(* IEC 61131-3 sources: RL_MAR/experiments/results/ablation/RL_MAR_DeepSeek-V3.2_full (part 2) *)

(* ---- med_62.st ---- *)
FUNCTION_BLOCK FB_PedestrianTrafficLight
VAR_INPUT
    pedBtnPress : BOOL;
END_VAR

VAR_OUTPUT
    carLightIsGreen : BOOL;
    pedLightIsGreen : BOOL;
    TimeCounter : INT;
END_VAR

VAR
    buttonPressedBefore : BOOL := FALSE;
    currentState : INT := 0;
    nextState : INT := 0;
END_VAR

CASE currentState OF
    0:
        carLightIsGreen := TRUE;
        pedLightIsGreen := FALSE;
        TimeCounter := 0;

        IF pedBtnPress AND NOT buttonPressedBefore THEN
            buttonPressedBefore := TRUE;
            nextState := 1;
        ELSE
            nextState := 0;
        END_IF;

    1:
        carLightIsGreen := FALSE;
        pedLightIsGreen := FALSE;
        TimeCounter := TimeCounter + 1;

        IF TimeCounter >= 10 THEN
            nextState := 2;
        ELSE
            nextState := 1;
        END_IF;

    2:
        carLightIsGreen := FALSE;
        pedLightIsGreen := TRUE;
        TimeCounter := TimeCounter + 1;

        IF TimeCounter >= 40 THEN
            nextState := 3;
        ELSE
            nextState := 2;
        END_IF;

    3:
        carLightIsGreen := FALSE;
        pedLightIsGreen := FALSE;
        TimeCounter := TimeCounter + 1;

        IF TimeCounter >= 50 THEN
            buttonPressedBefore := FALSE;
            nextState := 0;
        ELSE
            nextState := 3;
        END_IF;

    ELSE
        nextState := 0;
END_CASE;

currentState := nextState;

END_FUNCTION_BLOCK;

(* ---- med_63.st ---- *)
FUNCTION_BLOCK Automated_Parking_Controller
VAR_INPUT
    EntryGateSensor : BOOL; (* Sensor input for entry gate *)
    ExitGateSensor : BOOL; (* Sensor input for exit gate *)
    CarDetected : BOOL; (* Sensor input for car detection *)
END_VAR

VAR_OUTPUT
    ParkingSpaceNumber : INT := 0; (* Allocated parking space number *)
    RetrievalInProgress : BOOL := FALSE; (* Flag for car retrieval in progress *)
END_VAR

VAR
    ParkingSpaces : ARRAY[1..100] OF BOOL; (* Parking space status: TRUE=Occupied, FALSE=Available *)
    i : INT; (* Loop counter *)
    SpaceToRetrieve : INT := 0; (* Parking space number to retrieve *)
    RetrievalComplete : BOOL := FALSE; (* Internal flag for retrieval completion *)
END_VAR

METHOD MoveCarToExitGate : BOOL
VAR_INPUT
    SpaceNumber : INT;
END_VAR
BEGIN
    // Simulate car movement to exit gate
    // In a real system, this would control actuators, motors, etc.
    // For now, return TRUE to indicate successful movement
    MoveCarToExitGate := TRUE;
END_METHOD

// Main logic
IF NOT RetrievalInProgress THEN
    // Entry gate management
    IF EntryGateSensor THEN
        // Find first available parking space
        ParkingSpaceNumber := 0;
        FOR i := 1 TO 100 DO
            IF NOT ParkingSpaces[i] THEN
                ParkingSpaceNumber := i;
                ParkingSpaces[i] := TRUE;
                EXIT;
            END_IF;
        END_FOR;
    END_IF;
END_IF;

// Car retrieval management
IF CarDetected AND NOT RetrievalInProgress THEN
    RetrievalInProgress := TRUE;
    SpaceToRetrieve := ParkingSpaceNumber;
    RetrievalComplete := FALSE;
END_IF;

IF RetrievalInProgress THEN
    IF NOT RetrievalComplete THEN
        // Execute car movement to exit gate
        RetrievalComplete := MoveCarToExitGate(SpaceToRetrieve);
    ELSE
        // Wait for exit gate sensor to confirm car has left
        IF ExitGateSensor THEN
            // Mark parking space as available
            IF SpaceToRetrieve >= 1 AND SpaceToRetrieve <= 100 THEN
                ParkingSpaces[SpaceToRetrieve] := FALSE;
            END_IF;

            // Reset outputs
            ParkingSpaceNumber := 0;
            RetrievalInProgress := FALSE;
            SpaceToRetrieve := 0;
            RetrievalComplete := FALSE;
        END_IF;
    END_IF;
END_IF;

// Exit gate management (for normal exits without retrieval request)
IF ExitGateSensor AND NOT RetrievalInProgress AND ParkingSpaceNumber > 0 THEN
    // Mark current parking space as available
    IF ParkingSpaceNumber >= 1 AND ParkingSpaceNumber <= 100 THEN
        ParkingSpaces[ParkingSpaceNumber] := FALSE;
    END_IF;
    ParkingSpaceNumber := 0;
END_IF;

END_FUNCTION_BLOCK

(* ---- med_64.st ---- *)
FUNCTION_BLOCK BakeryOvenControl
VAR_INPUT
    TemperatureSensor : REAL; (* Sensor input for oven temperature *)
    HumiditySensor : REAL; (* Sensor input for oven humidity *)
END_VAR

VAR_OUTPUT
    HeatingElement : BOOL; (* Control signal for heating element *)
    CoolingElement : BOOL; (* Control signal for cooling element *)
    HumidityControl : BOOL; (* Control signal for humidity system *)
    DehumidityControl : BOOL; (* Control signal for dehumidification *)
END_VAR

VAR
    OvenTemperature : REAL := 180.0; (* Current oven temperature setpoint *)
    OvenHumidity : REAL := 60.0; (* Current oven humidity setpoint *)
    BakingTime : TIME := T#30M0S; (* Baking time setpoint *)
    OvenStatus : BOOL := FALSE; (* Oven status: TRUE=On, FALSE=Off *)
    HeatingThreshold : REAL := 2.0; (* Temperature control threshold *)
    HumidityThreshold : REAL := 5.0; (* Humidity control threshold *)
    TimerInstance : TON; (* Timer instance for 1-second decrement *)
    TimerPulse : BOOL := FALSE; (* Pulse for timer decrement *)
    InternalBakingTime : TIME := T#0S; (* Internal copy of baking time *)
END_VAR

(* Main logic body begins here *)

(* Timer for 1-second pulse generation *)
TimerInstance(IN := OvenStatus AND (InternalBakingTime > T#0S), PT := T#1S);
TimerPulse := TimerInstance.Q;

(* Decrement baking timer when oven is on and timer pulse is active *)
IF OvenStatus AND TimerPulse THEN
    IF InternalBakingTime > T#0S THEN
        InternalBakingTime := InternalBakingTime - T#1S;
    END_IF;
END_IF;

(* Reset internal timer when oven turns off *)
IF NOT OvenStatus THEN
    InternalBakingTime := BakingTime;
END_IF;

(* Main control logic - only active when oven is on and timer not expired *)
IF OvenStatus AND (InternalBakingTime > T#0S) THEN
    (* Temperature control logic *)
    IF TemperatureSensor < (OvenTemperature - HeatingThreshold) THEN
        HeatingElement := TRUE;
        CoolingElement := FALSE;
    ELSIF TemperatureSensor > (OvenTemperature + HeatingThreshold) THEN
        HeatingElement := FALSE;
        CoolingElement := TRUE;
    ELSE
        HeatingElement := FALSE;
        CoolingElement := FALSE;
    END_IF;

    (* Humidity control logic *)
    IF HumiditySensor < (OvenHumidity - HumidityThreshold) THEN
        HumidityControl := TRUE;
        DehumidityControl := FALSE;
    ELSIF HumiditySensor > (OvenHumidity + HumidityThreshold) THEN
        HumidityControl := FALSE;
        DehumidityControl := TRUE;
    ELSE
        HumidityControl := FALSE;
        DehumidityControl := FALSE;
    END_IF;

(* Oven off or timer expired - turn off all outputs *)
ELSE
    HeatingElement := FALSE;
    CoolingElement := FALSE;
    HumidityControl := FALSE;
    DehumidityControl := FALSE;

    (* Auto-shutdown when timer expires *)
    IF (InternalBakingTime <= T#0S) AND OvenStatus THEN
        OvenStatus := FALSE;
    END_IF;
END_IF;

END_FUNCTION_BLOCK;

(* ---- med_65.st ---- *)
FUNCTION_BLOCK TheaterControl
VAR_INPUT
    StartButton : BOOL; (* Input for starting a performance *)
    StopButton : BOOL; (* Input for stopping a performance *)
    SceneNumber : INT; (* Input for selecting the scene or act *)
END_VAR

VAR_OUTPUT
    LightingControl : BOOL; (* Output for controlling lighting *)
    SoundControl : BOOL; (* Output for controlling sound *)
    PerformanceInProgress : BOOL; (* Indicator for an ongoing performance *)
END_VAR

VAR
    CurrentState : INT := 1; (* 1=IDLE, 2=ACTIVE, 3=STOP *)
    NextState : INT;
END_VAR

(* State Machine Logic *)
CASE CurrentState OF
    1: (* IDLE State *)
        LightingControl := FALSE;
        SoundControl := FALSE;
        PerformanceInProgress := FALSE;

        IF StopButton THEN
            NextState := 3;
        ELSIF StartButton AND NOT PerformanceInProgress THEN
            IF (SceneNumber >= 1) AND (SceneNumber <= 3) THEN
                NextState := 2;
            ELSE
                NextState := 3;
            END_IF;
        ELSE
            NextState := 1;
        END_IF;

    2: (* ACTIVE State *)
        LightingControl := TRUE;
        SoundControl := TRUE;
        PerformanceInProgress := TRUE;

        IF StopButton THEN
            NextState := 3;
        ELSE
            NextState := 2;
        END_IF;

    3: (* STOP State *)
        LightingControl := FALSE;
        SoundControl := FALSE;
        PerformanceInProgress := FALSE;
        NextState := 1;

END_CASE;

(* State Transition *)
CurrentState := NextState;

END_FUNCTION_BLOCK;

(* ---- med_66.st ---- *)
FUNCTION_BLOCK ElevatorControl
VAR_INPUT
    CurrentPos : INT;
    RequestedPos : INT;
    ButtonPressed : BOOL;
END_VAR

VAR_OUTPUT
    MotorMovingUp : BOOL;
    MotorMovingDown : BOOL;
    DoorIsOpen : BOOL;
END_VAR

VAR
    bMovementInitiated : BOOL := FALSE;
END_VAR

(* Main logic body begins here *)

(* Reset outputs on each cycle *)
MotorMovingUp := FALSE;
MotorMovingDown := FALSE;
DoorIsOpen := FALSE;

(* Handle button press to initiate movement *)
IF ButtonPressed THEN
    bMovementInitiated := TRUE;
    DoorIsOpen := FALSE;
END_IF;

(* Determine movement direction and handle state transitions *)
IF bMovementInitiated THEN
    IF CurrentPos < RequestedPos THEN
        (* Move up *)
        MotorMovingUp := TRUE;
        MotorMovingDown := FALSE;
        DoorIsOpen := FALSE;
    ELSIF CurrentPos > RequestedPos THEN
        (* Move down *)
        MotorMovingUp := FALSE;
        MotorMovingDown := TRUE;
        DoorIsOpen := FALSE;
    ELSE
        (* Reached destination *)
        MotorMovingUp := FALSE;
        MotorMovingDown := FALSE;
        DoorIsOpen := TRUE;
        bMovementInitiated := FALSE;
    END_IF;
ELSE
    (* Stationary at requested floor *)
    IF CurrentPos = RequestedPos THEN
        DoorIsOpen := TRUE;
    END_IF;
END_IF;

END_FUNCTION_BLOCK;

(* ---- med_67.st ---- *)
FUNCTION_BLOCK FB_FactorialCalculator
VAR_INPUT
    X : INT;
END_VAR

VAR_OUTPUT
    FactorialResult : INT;
    FactorialGoodResult : INT;
END_VAR

VAR
    tempGoodResult : INT;
    tempResult : INT;
END_VAR

// Main logic
IF (X >= -3) AND (X <= 3) THEN
    // Calculate FactorialGoodResult = X * X * X * X
    tempGoodResult := X * X;
    tempGoodResult := tempGoodResult * X;
    tempGoodResult := tempGoodResult * X;
    FactorialGoodResult := tempGoodResult;

    // Calculate FactorialResult
    IF FactorialGoodResult > 1 THEN
        tempResult := FactorialGoodResult - 1;
        FactorialResult := FactorialGoodResult * tempResult;
    ELSE
        FactorialResult := FactorialGoodResult;
    END_IF;
ELSE
    // X is outside range [-3, 3]
    FactorialGoodResult := 0;
    FactorialResult := 1;
END_IF;
END_FUNCTION_BLOCK

(* ---- med_68.st ---- *)
FUNCTION_BLOCK SignalControl
VAR_INPUT
    Int1 : BOOL;
    Int2 : BOOL;
    Int3 : BOOL;
    Int4 : BOOL;
    Int5 : BOOL;
    Int6 : BOOL;
    Int7 : BOOL;
    Int8 : BOOL;
    IntAn1 : UINT;
    IntAn2 : UINT;
    IntAn3 : UINT;
    IntAn4 : UINT;
    IntAn5 : UINT;
    IntAn6 : UINT;
    IntAn7 : UINT;
    IntAn8 : UINT;
    Marca2 : BOOL;
END_VAR

VAR_OUTPUT
    Out1 : BOOL;
    Out2 : BOOL;
    Out3 : BOOL;
    Out4 : BOOL;
    Out5 : BOOL;
    Out6 : BOOL;
    Out7 : BOOL;
    Out8 : BOOL;
    OutAn1 : UINT;
    OutAn2 : UINT;
    OutAn3 : UINT;
    OutAn4 : UINT;
    OutAn5 : UINT;
    OutAn6 : UINT;
    OutAn7 : UINT;
    OutAn8 : UINT;
END_VAR

VAR
    Marca1 : BOOL;
    GT51_OUT : BOOL;
    GT56_OUT : BOOL;
    GT57_OUT : BOOL;
    GT62_OUT : BOOL;
END_VAR

    (* Logic for Marca1 flag *)
    IF NOT Marca2 AND ((Marca1 OR NOT Out1) AND Int1) THEN
        Marca1 := TRUE;
    ELSE
        Marca1 := FALSE;
    END_IF;

    (* Latch behavior for Out1 *)
    IF NOT Marca2 AND (Marca1 OR Out1) THEN
        Out1 := TRUE;
    ELSE
        Out1 := FALSE;
    END_IF;

    (* Direct Boolean pass-through *)
    Out2 := Int2;
    Out3 := Int3;
    Out4 := Int4;

    (* Direct unsigned integer pass-through *)
    OutAn1 := IntAn1;
    OutAn2 := IntAn2;
    OutAn3 := IntAn3;
    OutAn4 := IntAn4;

    (* Conditional outputs with comparison results *)
    GT51_OUT := (IntAn5 > 1000);
    GT56_OUT := (IntAn6 > 1000);
    GT57_OUT := (IntAn7 > 1000);
    GT62_OUT := (IntAn8 > 1000);

    (* Conditional output logic for Out5 *)
    IF GT51_OUT AND NOT Int5 THEN
        Out5 := TRUE;
    ELSE
        Out5 := FALSE;
    END_IF;

    (* Conditional output logic for Out6 *)
    IF GT56_OUT AND NOT Int6 THEN
        Out6 := TRUE;
    ELSE
        Out6 := FALSE;
    END_IF;

    (* Conditional output logic for Out7 *)
    IF GT57_OUT AND NOT Int7 THEN
        Out7 := TRUE;
    ELSE
        Out7 := FALSE;
    END_IF;

    (* Conditional output logic for Out8 *)
    IF GT62_OUT AND NOT Int8 THEN
        Out8 := TRUE;
    ELSE
        Out8 := FALSE;
    END_IF;

    (* Pass through remaining analog values *)
    OutAn5 := IntAn5;
    OutAn6 := IntAn6;
    OutAn7 := IntAn7;
    OutAn8 := IntAn8;

END_FUNCTION_BLOCK;

(* ---- med_69.st ---- *)
FUNCTION_BLOCK FB_ValueOut
VAR_INPUT
    valueIn : INT;
    conf : UINT;
END_VAR

VAR_OUTPUT
    ValueOut : INT;
END_VAR

VAR
    tempResult : INT;
END_VAR

(* Main logic body *)
CASE conf OF
    1, 2:
        tempResult := valueIn / 10;
        IF tempResult < 0 THEN
            ValueOut := 0;
        ELSE
            ValueOut := tempResult;
        END_IF;

    3:
        IF valueIn = 0 THEN
            ValueOut := 0;
        ELSIF valueIn = 300 THEN
            ValueOut := 163;
        ELSIF valueIn = 600 THEN
            ValueOut := 331;
        ELSE
            ValueOut := 0;
        END_IF;

    6, 7:
        IF valueIn = 100 THEN
            ValueOut := 319;
        ELSE
            ValueOut := 0;
        END_IF;

    ELSE
        ValueOut := 0;
END_CASE;

END_FUNCTION_BLOCK;

(* ---- med_70.st ---- *)
FUNCTION_BLOCK EggIncubatorControl
VAR_INPUT
    StartButton : BOOL; (* Input for starting the incubation process *)
    StopButton : BOOL; (* Input for stopping the incubation process *)
    TemperatureSensor : REAL; (* Input for temperature reading in °C *)
    HumiditySensor : REAL; (* Input for humidity reading in % *)
END_VAR

VAR_OUTPUT
    HeatingElement : BOOL; (* Output for controlling the heating element *)
    Humidifier : BOOL; (* Output for controlling the humidifier *)
    EggTurningMotor : BOOL; (* Output for controlling the egg turning motor *)
    IncubationInProgress : BOOL; (* Indicator for an ongoing incubation process *)
END_VAR

VAR
    TargetTemperature : REAL; (* Target temperature in °C *)
    TargetHumidity : REAL; (* Target humidity in % *)
    TurnIntervalSeconds : INT; (* Interval for turning eggs (1 hour in seconds) *)
    TurnTimerSeconds : INT; (* Timer for egg turning cycle in seconds *)
END_VAR

(* Initialize control parameters *)
TargetTemperature := 37.5;
TargetHumidity := 50.0;
TurnIntervalSeconds := 3600;

(* Start/Stop Control *)
IF StartButton AND NOT IncubationInProgress THEN
    IncubationInProgress := TRUE;
END_IF;

IF StopButton THEN
    IncubationInProgress := FALSE;
    HeatingElement := FALSE;
    Humidifier := FALSE;
    EggTurningMotor := FALSE;
    TurnTimerSeconds := 0;
END_IF;

(* Temperature Control *)
IF TemperatureSensor < TargetTemperature THEN
    HeatingElement := TRUE;
ELSE
    HeatingElement := FALSE;
END_IF;

(* Humidity Control *)
IF HumiditySensor < TargetHumidity THEN
    Humidifier := TRUE;
ELSE
    Humidifier := FALSE;
END_IF;

(* Egg Turning Cycle *)
IF IncubationInProgress THEN
    TurnTimerSeconds := TurnTimerSeconds + 1;
    IF TurnTimerSeconds >= TurnIntervalSeconds THEN
        EggTurningMotor := NOT EggTurningMotor;
        TurnTimerSeconds := 0;
    END_IF;
END_IF;

END_FUNCTION_BLOCK;

(* ---- med_71.st ---- *)
FUNCTION_BLOCK FB_Fibonacci_Calculator
VAR_INPUT
    N : DINT := 5;
END_VAR
VAR_OUTPUT
    O : DINT := 1;
END_VAR
VAR
    F1 : DINT := 1;
    F2 : DINT := 1;
    CNT : DINT := 2;
    Temp : DINT;
END_VAR

// Handle edge cases: N <= 2 returns 1
IF N <= 2 THEN
    O := 1;
    RETURN;
END_IF;

// Initialize for calculation
F1 := 1;
F2 := 1;
CNT := 2;

// Calculate Fibonacci sequence up to N-th term
WHILE CNT < N DO
    // Check for potential overflow before calculation
    IF (F1 > 32767 - F2) THEN
        // Saturation: if sum would exceed 32767, saturate to 32767
        O := 32767;
        RETURN;
    END_IF;

    // Calculate next Fibonacci number
    Temp := F1 + F2;
    F1 := F2;
    F2 := Temp;
    CNT := CNT + 1;
END_WHILE;

// Set output to the N-th Fibonacci number
O := F2;

// Final saturation check (in case F2 already exceeded 32767)
IF O > 32767 THEN
    O := 32767;
END_IF;

END_FUNCTION_BLOCK

(* ---- med_72.st ---- *)
FUNCTION_BLOCK DigitalSignageManagement
VAR_INPUT
    DisplayLocations : ARRAY[1..10] OF BOOL;
    ContentSource : ARRAY[1..10] OF INT;
END_VAR

VAR_OUTPUT
    CurrentContent : ARRAY[1..10] OF INT;
END_VAR

VAR
    i : INT;
END_VAR

FOR i := 1 TO 10 DO
    IF DisplayLocations[i] THEN
        CASE ContentSource[i] OF
            1:
                CurrentContent[i] := 1;
            2:
                CurrentContent[i] := 2;
            3:
                CurrentContent[i] := 3;
            ELSE
                CurrentContent[i] := 0;
        END_CASE;
    ELSE
        CurrentContent[i] := 0;
    END_IF;
END_FOR;

END_FUNCTION_BLOCK;

(* ---- med_73.st ---- *)
FUNCTION_BLOCK RoboticWeldingSystem
    VAR_INPUT
        RobotArm1Ready : BOOL; (* Input for robot arm 1 ready status *)
        RobotArm2Ready : BOOL; (* Input for robot arm 2 ready status *)
        WeldingGunReady : BOOL; (* Input for welding gun ready status *)
        StartButton : BOOL; (* Input for start button press *)
        StopButton : BOOL; (* Input for stop button press *)
    END_VAR

    VAR_OUTPUT
        WeldingTrigger : BOOL; (* Output to trigger welding *)
        WeldingComplete : BOOL; (* Output indicating welding completion *)
    END_VAR

    VAR
        weldingActive : BOOL;
    END_VAR

    IF StopButton THEN
        weldingActive := FALSE;
        WeldingTrigger := FALSE;
        WeldingComplete := TRUE;
    ELSE
        IF NOT weldingActive AND RobotArm1Ready AND RobotArm2Ready AND WeldingGunReady AND StartButton THEN
            weldingActive := TRUE;
            WeldingTrigger := TRUE;
            WeldingComplete := FALSE;
        ELSIF weldingActive THEN
            WeldingTrigger := TRUE;
            WeldingComplete := FALSE;
        ELSE
            WeldingTrigger := FALSE;
            WeldingComplete := TRUE;
        END_IF;
    END_IF;
END_FUNCTION_BLOCK

(* ---- med_74.st ---- *)
FUNCTION_BLOCK TrafficManagementSystem
VAR_INPUT
    VehicleCount1 : INT; (* Input for vehicle count at intersection 1 *)
    VehicleCount2 : INT; (* Input for vehicle count at intersection 2 *)
    VehicleCount3 : INT; (* Input for vehicle count at intersection 3 *)
    VehicleCount4 : INT; (* Input for vehicle count at intersection 4 *)
END_VAR

VAR_OUTPUT
    TrafficLight1 : BOOL; (* Output for traffic light at intersection 1 *)
    TrafficLight2 : BOOL; (* Output for traffic light at intersection 2 *)
    TrafficLight3 : BOOL; (* Output for traffic light at intersection 3 *)
    TrafficLight4 : BOOL; (* Output for traffic light at intersection 4 *)
END_VAR

VAR
    (* No internal variables needed for this simplified implementation *)
END_VAR

(* Main logic for intersection pair 1 (Intersections 1 and 2) *)
IF VehicleCount1 > VehicleCount2 THEN
    TrafficLight1 := TRUE;
    TrafficLight2 := FALSE;
ELSIF VehicleCount1 < VehicleCount2 THEN
    TrafficLight1 := FALSE;
    TrafficLight2 := TRUE;
ELSE
    TrafficLight1 := FALSE;
    TrafficLight2 := FALSE;
END_IF;

(* Main logic for intersection pair 2 (Intersections 3 and 4) *)
IF VehicleCount3 > VehicleCount4 THEN
    TrafficLight3 := TRUE;
    TrafficLight4 := FALSE;
ELSIF VehicleCount3 < VehicleCount4 THEN
    TrafficLight3 := FALSE;
    TrafficLight4 := TRUE;
ELSE
    TrafficLight3 := FALSE;
    TrafficLight4 := FALSE;
END_IF;

END_FUNCTION_BLOCK;

(* ---- med_75.st ---- *)
FUNCTION_BLOCK HomeBrewingSystem
VAR_INPUT
    TemperatureSensor : REAL; (* Input for temperature measurement (°C) *)
    WaterFlowSensor : REAL; (* Input for water flow measurement (L/min) *)
    BrewingStartTime : TIME; (* Input for brewing process start time *)
    BrewingDuration : TIME; (* Input for total brewing duration *)
END_VAR

VAR_OUTPUT
    HeatingElement : BOOL; (* Output to control heating element *)
    AgitationMotor : BOOL; (* Output to control agitation motor *)
    HopsDispenser : BOOL; (* Output to control hops dispenser *)
    FermentationTank : BOOL; (* Output to control fermentation tank *)
END_VAR

VAR
    ElapsedTime : TIME;
    HopsTriggerTime : TIME := T#5h;
    FermentationTriggerTime : TIME := T#48h;
END_VAR

(* Main logic body *)
ElapsedTime := BrewingDuration;

(* Temperature control: heating element ON when temperature is below 65°C *)
HeatingElement := TemperatureSensor < 65.0;

(* Agitation motor control: motor ON when water flow exceeds 0.5 L/min *)
AgitationMotor := WaterFlowSensor > 0.5;

(* Hops dispenser: activate after 5 hours of brewing *)
HopsDispenser := ElapsedTime >= HopsTriggerTime;

(* Fermentation tank transfer: activate after 48 hours of brewing *)
FermentationTank := ElapsedTime >= FermentationTriggerTime;

END_FUNCTION_BLOCK;

(* ---- med_76.st ---- *)
FUNCTION_BLOCK MultimediaArtInstallationControl
VAR_INPUT
    MotionSensor : BOOL; (* Motion detection input *)
    AudioTrack : BOOL; (* Selected audio track *)
    VisualContent : BOOL; (* Selected visual content *)
END_VAR

VAR_OUTPUT
    LightingControl : BOOL; (* Lighting control output *)
    AudioControl : BOOL; (* Audio playback control *)
    VisualControl : BOOL; (* Visual display control *)
    ActivationTimer : INT; (* Timer for activation duration *)
END_VAR

VAR
    bMotionDetectedPrev : BOOL; (* Previous state of motion sensor *)
    bElementsActive : BOOL; (* State of all multimedia elements *)
END_VAR

(* Main logic *)
IF MotionSensor THEN
    (* Motion detected: activate all elements *)
    LightingControl := TRUE;
    AudioControl := AudioTrack; (* Only activate if audio track is selected *)
    VisualControl := VisualContent; (* Only activate if visual content is selected *)
    bElementsActive := TRUE;

    (* Increment activation timer up to 300 seconds *)
    IF ActivationTimer < 300 THEN
        ActivationTimer := ActivationTimer + 1;
    END_IF;

    (* Store current motion state for edge detection *)
    bMotionDetectedPrev := TRUE;

ELSE
    (* No motion detected: deactivate all elements *)
    LightingControl := FALSE;
    AudioControl := FALSE;
    VisualControl := FALSE;
    bElementsActive := FALSE;

    (* Reset timer when no motion is detected *)
    ActivationTimer := 0;

    (* Store current motion state for edge detection *)
    bMotionDetectedPrev := FALSE;
END_IF;

(* Safety protocol: Ensure elements are only active when motion is detected *)
IF NOT MotionSensor AND bElementsActive THEN
    LightingControl := FALSE;
    AudioControl := FALSE;
    VisualControl := FALSE;
    bElementsActive := FALSE;
    ActivationTimer := 0;
END_IF;

END_FUNCTION_BLOCK

(* ---- med_77.st ---- *)
FUNCTION_BLOCK OutdoorLEDLightingControl
VAR_INPUT
    AmbientLight : REAL; (* 环境光传感器输入 *)
    MotionSensor : BOOL; (* 运动传感器输入 *)
    EnergySaving : BOOL; (* 节能模式开关 *)
END_VAR

VAR_OUTPUT
    Light : BOOL; (* LED照明控制输出 *)
    EnergyMode : BOOL; (* 节能模式状态输出 *)
END_VAR

VAR
    (* No internal variables needed for this simple logic *)
END_VAR

(* Main logic body *)
IF MotionSensor THEN
    (* Motion Detection Override: Highest priority *)
    Light := TRUE;
    EnergyMode := FALSE; (* Override: deactivate energy-saving mode *)
ELSE
    (* No motion detected: evaluate ambient light and energy-saving mode *)
    IF (AmbientLight < 50.0) AND (NOT EnergySaving) THEN
        Light := TRUE;
    ELSE
        Light := FALSE;
    END_IF;

    (* Energy mode status reflects the input *)
    EnergyMode := EnergySaving;
END_IF;

END_FUNCTION_BLOCK;

(* ---- med_78.st ---- *)
FUNCTION_BLOCK RetractableRoofControl
    VAR_INPUT
        RainSensor : BOOL; (* Rain detection *)
        WindSensor : BOOL; (* Wind detection *)
        TemperatureSensor : REAL; (* Temperature input *)
    END_VAR

    VAR_OUTPUT
        RoofMotor : BOOL; (* Motor control *)
    END_VAR

    VAR
        TemperatureThreshold : REAL := 20.0;
    END_VAR

    (* Main logic body begins here *)
    IF RainSensor AND WindSensor THEN
        RoofMotor := TRUE;
    ELSIF RainSensor THEN
        RoofMotor := TRUE;
    ELSIF TemperatureSensor < TemperatureThreshold THEN
        RoofMotor := TRUE;
    ELSE
        RoofMotor := FALSE;
    END_IF;

END_FUNCTION_BLOCK;

(* ---- med_79.st ---- *)
FUNCTION_BLOCK CapsuleFillingMachineControl
VAR_INPUT
    CapsuleWeight : REAL;        (* Current capsule weight *)
    TargetWeight : REAL;         (* Target weight to achieve *)
    CapsuleInPosition : BOOL;    (* Capsule position sensor *)
    HopperEmpty : BOOL;          (* Hopper empty sensor *)
END_VAR
VAR_OUTPUT
    FeederMotor : BOOL;          (* Feeder motor control *)
    FillingMotor : BOOL;         (* Filling motor control *)
    ConveyorMotor : BOOL;        (* Conveyor motor control *)
    FillingInProgress : BOOL;    (* Filling status *)
    ErrorCode : INT;             (* Error indication: 0=OK, 1=CapsuleNotDetected, 2=FillingTimeout *)
END_VAR
VAR
    (* State machine *)
    CurrentState : INT := 0;     (* 0=IDLE, 1=CONVEYING, 2=FILLING, 3=CONVEYING_OUT *)

    (* Timers *)
    ConveyorTimer : TON;
    FillingTimer : TON;
    ConveyOutTimer : TON;

    (* Timing parameters *)
    ConveyorTime : TIME := T#2S;
    MaxFillingTime : TIME := T#10S;
    ConveyOutTime : TIME := T#1S;

    (* Error detection *)
    CapsuleDetectTimeout : TON;
    CapsuleDetectTime : TIME := T#5S;

    (* Filling control *)
    WeightTolerance : REAL := 0.1;
    FillingSpeed : REAL := 0.0;
    LastCapsuleWeight : REAL := 0.0;

    (* Internal flags *)
    CapsuleDetected : BOOL := FALSE;
    FillingComplete : BOOL := FALSE;
    ErrorFlag : BOOL := FALSE;
END_VAR

(* Safety Check: Hopper Empty *)
IF HopperEmpty THEN
    FeederMotor := FALSE;
    FillingMotor := FALSE;
    ConveyorMotor := FALSE;
    FillingInProgress := FALSE;
    ErrorCode := 0;
    CurrentState := 0;
    RETURN;
END_IF;

(* Weight Validation: Initial Check *)
IF CapsuleWeight >= TargetWeight AND NOT FillingInProgress THEN
    FeederMotor := FALSE;
    FillingMotor := FALSE;
    ConveyorMotor := FALSE;
    FillingInProgress := FALSE;
    ErrorCode := 0;
    CurrentState := 0;
    RETURN;
END_IF;

(* State Machine Execution *)
CASE CurrentState OF
    0: (* IDLE *)
        FeederMotor := TRUE;
        FillingMotor := FALSE;
        ConveyorMotor := FALSE;
        FillingInProgress := FALSE;
        FillingComplete := FALSE;
        ErrorFlag := FALSE;
        ErrorCode := 0;

        (* Reset timers *)
        ConveyorTimer(IN:=FALSE, PT:=ConveyorTime);
        FillingTimer(IN:=FALSE, PT:=MaxFillingTime);
        ConveyOutTimer(IN:=FALSE, PT:=ConveyOutTime);
        CapsuleDetectTimeout(IN:=FALSE, PT:=CapsuleDetectTime);

        (* Check for capsule detection *)
        IF CapsuleInPosition THEN
            CapsuleDetected := TRUE;
            CurrentState := 1; (* Move to CONVEYING state *)
            ConveyorTimer(IN:=TRUE, PT:=ConveyorTime);
        ELSE
            (* Start capsule detection timeout *)
            CapsuleDetectTimeout(IN:=TRUE, PT:=CapsuleDetectTime);
            IF CapsuleDetectTimeout.Q THEN
                ErrorCode := 1; (* CapsuleNotDetected *)
                ErrorFlag := TRUE;
            END_IF;
        END_IF;

    1: (* CONVEYING *)
        FeederMotor := TRUE;
        FillingMotor := FALSE;
        ConveyorMotor := TRUE;
        FillingInProgress := FALSE;

        (* Run conveyor timer *)
        ConveyorTimer(IN:=TRUE, PT:=ConveyorTime);

        IF ConveyorTimer.Q THEN
            (* Conveying complete, start filling *)
            CurrentState := 2; (* Move to FILLING state *)
            FillingTimer(IN:=TRUE, PT:=MaxFillingTime);
            FillingInProgress := TRUE;
            LastCapsuleWeight := CapsuleWeight;
        END_IF;

    2: (* FILLING *)
        FeederMotor := TRUE;
        ConveyorMotor := FALSE;
        FillingInProgress := TRUE;

        (* Simple proportional filling control *)
        IF TargetWeight > CapsuleWeight THEN
            (* Calculate filling speed based on weight difference *)
            FillingSpeed := (TargetWeight - CapsuleWeight) / TargetWeight;

            (* Limit filling speed between 0.1 and 1.0 *)
            IF FillingSpeed < 0.1 THEN
                FillingSpeed := 0.1;
            ELSIF FillingSpeed > 1.0 THEN
                FillingSpeed := 1.0;
            END_IF;

            (* Control filling motor with speed-based duty cycle *)
            FillingMotor := TRUE;
        ELSE
            FillingMotor := FALSE;
            FillingComplete := TRUE;
        END_IF;

        (* Check if target weight is reached within tolerance *)
        IF CapsuleWeight >= (TargetWeight - WeightTolerance) THEN
            FillingMotor := FALSE;
            FillingComplete := TRUE;
        END_IF;

        (* Check for filling timeout *)
        FillingTimer(IN:=TRUE, PT:=MaxFillingTime);
        IF FillingTimer.Q AND NOT FillingComplete THEN
            ErrorCode := 2; (* FillingTimeout *)
            ErrorFlag := TRUE;
            CurrentState := 0; (* Return to IDLE *)
        END_IF;

        (* Move to next state when filling is complete *)
        IF FillingComplete AND NOT ErrorFlag THEN
            CurrentState := 3; (* Move to CONVEYING_OUT state *)
            ConveyOutTimer(IN:=TRUE, PT:=ConveyOutTime);
        END_IF;

    3: (* CONVEYING_OUT *)
        FeederMotor := TRUE;
        FillingMotor := FALSE;
        ConveyorMotor := TRUE;
        FillingInProgress := FALSE;

        (* Run conveyor out timer *)
        ConveyOutTimer(IN:=TRUE, PT:=ConveyOutTime);

        IF ConveyOutTimer.Q THEN
            (* Conveying out complete, return to IDLE *)
            CurrentState := 0;
            CapsuleDetected := FALSE;
            FillingComplete := FALSE;
        END_IF;

END_CASE;

(* Update timers *)
ConveyorTimer();
FillingTimer();
ConveyOutTimer();
CapsuleDetectTimeout();

END_FUNCTION_BLOCK

(* ---- med_80.st ---- *)
FUNCTION_BLOCK DoughMixerControl
    VAR_INPUT
        IngredientsDetected : BOOL;
    END_VAR

    VAR_OUTPUT
        MixingInProgress : BOOL;
    END_VAR

    VAR
        MixingTimeElapsed : TIME;
        MixingTimeLimit : TIME := T#5S;
        LastIngredientsDetected : BOOL;
    END_VAR

    IF IngredientsDetected AND NOT LastIngredientsDetected THEN
        MixingInProgress := TRUE;
        MixingTimeElapsed := T#0S;
    ELSIF NOT IngredientsDetected OR MixingTimeElapsed >= MixingTimeLimit THEN
        MixingInProgress := FALSE;
    END_IF;

    IF MixingInProgress THEN
        MixingTimeElapsed := MixingTimeElapsed + T#1S;
    END_IF;

    LastIngredientsDetected := IngredientsDetected;
END_FUNCTION_BLOCK;

(* ---- med_81.st ---- *)
FUNCTION_BLOCK SolarPanelTracking
    VAR_INPUT
        CurrentTime : TIME;
        SolarIntensity : REAL;
    END_VAR

    VAR_OUTPUT
        PanelAngle : REAL;
    END_VAR

    VAR
        SunriseTime : TIME := T#6H;
        NoonTime : TIME := T#12H;
        SunsetTime : TIME := T#18H;
        MorningAngle : REAL := 30.0;
        NoonAngle : REAL := 60.0;
        EveningAngle : REAL := 30.0;
    END_VAR

    (* Main logic body *)
    IF SolarIntensity >= 90.0 THEN
        PanelAngle := NoonAngle;
    ELSE
        IF (CurrentTime < SunriseTime) OR (CurrentTime >= SunsetTime) THEN
            PanelAngle := 0.0;
        ELSIF (CurrentTime >= SunriseTime) AND (CurrentTime < NoonTime) THEN
            PanelAngle := MorningAngle;
        ELSIF (CurrentTime >= NoonTime) AND (CurrentTime < SunsetTime) THEN
            PanelAngle := EveningAngle;
        END_IF;
    END_IF;
END_FUNCTION_BLOCK;

(* ---- med_82.st ---- *)
FUNCTION_BLOCK PetFeederControl
VAR_INPUT
    CurrentTime : TIME; (* Current system time input *)
END_VAR

VAR_OUTPUT
    FoodDispense : BOOL; (* Food dispenser control signal *)
END_VAR

VAR
    FeedTime1 : TIME := T#8H0M0S; (* First feeding time - 8:00 AM *)
    FeedTime2 : TIME := T#12H0M0S; (* Second feeding time - 12:00 PM *)
    FeedTime3 : TIME := T#18H0M0S; (* Third feeding time - 6:00 PM *)
    FoodAmount : INT := 50; (* Amount of food to dispense in grams *)
END_VAR

(* Main dispensing logic *)
FoodDispense := (CurrentTime >= FeedTime1 AND CurrentTime < FeedTime1 + T#30S) OR
                (CurrentTime >= FeedTime2 AND CurrentTime < FeedTime2 + T#30S) OR
                (CurrentTime >= FeedTime3 AND CurrentTime < FeedTime3 + T#30S);

END_FUNCTION_BLOCK;

(* ---- med_83.st ---- *)
FUNCTION_BLOCK AmusementRideControl
    VAR_INPUT
        StartButton : BOOL; (* Start button input *)
        StopButton : BOOL; (* Emergency stop button input *)
        SpeedSensor : REAL; (* Speed sensor input (RPM) *)
        SafetySensor : BOOL; (* Safety sensor status *)
    END_VAR

    VAR_OUTPUT
        MotorOn : BOOL := FALSE; (* Motor control output *)
        BrakeOn : BOOL := TRUE; (* Brake control output *)
    END_VAR

    VAR
        SpeedLimit : REAL := 60.0; (* Maximum allowed speed in RPM *)
    END_VAR

    (* Main logic body *)
    IF StopButton THEN
        (* Emergency Stop - Highest Priority *)
        MotorOn := FALSE;
        BrakeOn := TRUE;
    ELSIF StartButton AND (NOT StopButton) AND (SpeedSensor <= SpeedLimit) AND SafetySensor THEN
        (* Start Condition - All Conditions Met *)
        MotorOn := TRUE;
        BrakeOn := FALSE;
    ELSE
        (* Default State - Fail-Safe *)
        MotorOn := FALSE;
        BrakeOn := TRUE;
    END_IF;

    (* Runtime Safety Monitoring *)
    IF MotorOn AND ((SpeedSensor > SpeedLimit) OR (NOT SafetySensor)) THEN
        MotorOn := FALSE;
        BrakeOn := TRUE;
    END_IF;

END_FUNCTION_BLOCK;

(* ---- med_84.st ---- *)
FUNCTION_BLOCK ParcelSortingSystem
    VAR_INPUT
        ParcelSizeSensor : REAL; (* Sensor input for parcel size *)
        DestinationCodeSensor : INT; (* Destination code: 1=A, 2=B *)
    END_VAR

    VAR_OUTPUT
        ConveyorBeltMotor : BOOL; (* Output for conveyor belt motor: TRUE=On, FALSE=Off *)
        SortingGate1 : BOOL; (* Output for sorting gate 1: TRUE=Open, FALSE=Closed *)
        SortingGate2 : BOOL; (* Output for sorting gate 2: TRUE=Open, FALSE=Closed *)
    END_VAR

    VAR
        bSizeValid : BOOL;
        bDestValid : BOOL;
        bIsLarge : BOOL;
        rSizeThreshold : REAL := 50.0;
    END_VAR

    (* Main logic body begins here *)

    (* Input validation *)
    bSizeValid := ParcelSizeSensor > 0.0;
    bDestValid := (DestinationCodeSensor = 1) OR (DestinationCodeSensor = 2);

    (* Size classification *)
    IF ParcelSizeSensor >= rSizeThreshold THEN
        bIsLarge := TRUE;
    ELSE
        bIsLarge := FALSE;
    END_IF;

    (* Main control logic *)
    IF bSizeValid AND bDestValid THEN
        ConveyorBeltMotor := TRUE;

        CASE DestinationCodeSensor OF
            1: (* Destination A *)
                IF bIsLarge THEN
                    SortingGate1 := TRUE;
                    SortingGate2 := FALSE;
                ELSE
                    SortingGate1 := FALSE;
                    SortingGate2 := TRUE;
                END_IF;

            2: (* Destination B *)
                IF bIsLarge THEN
                    SortingGate1 := TRUE;
                    SortingGate2 := FALSE;
                ELSE
                    SortingGate1 := FALSE;
                    SortingGate2 := FALSE;
                END_IF;

            ELSE
                SortingGate1 := FALSE;
                SortingGate2 := FALSE;
        END_CASE;
    ELSE
        (* Invalid input - stop conveyor and close all gates *)
        ConveyorBeltMotor := FALSE;
        SortingGate1 := FALSE;
        SortingGate2 := FALSE;
    END_IF;

END_FUNCTION_BLOCK;

(* ---- med_85.st ---- *)
FUNCTION_BLOCK ShredderControl
    VAR_INPUT
        StartButton : BOOL;
        StopButton : BOOL;
        EmergencyStop : BOOL;
        MaterialInFeed : BOOL;
        JammedSensor : BOOL;
    END_VAR

    VAR_OUTPUT
        MotorControl : BOOL;
        SafetyRelay : BOOL;
    END_VAR

    VAR
        bMotorRunning : BOOL;
    END_VAR

    (* Highest Priority: Emergency Stop and Jam Detection *)
    IF EmergencyStop OR JammedSensor THEN
        MotorControl := FALSE;
        SafetyRelay := FALSE;
        bMotorRunning := FALSE;
    ELSE
        (* Normal Operation Logic *)
        IF (StartButton OR MaterialInFeed) AND NOT bMotorRunning THEN
            bMotorRunning := TRUE;
        ELSIF StopButton THEN
            bMotorRunning := FALSE;
        END_IF;

        (* Motor Control Output *)
        MotorControl := bMotorRunning;

        (* Safety Relay Output - Active during normal operation when motor is running or ready to run *)
        SafetyRelay := bMotorRunning OR ((StartButton OR MaterialInFeed) AND NOT StopButton);
    END_IF;

END_FUNCTION_BLOCK;

(* ---- med_86.st ---- *)
FUNCTION_BLOCK FruitJuicingBottling
    VAR_INPUT
        StartButton : BOOL; (* Input for starting the process *)
        StopButton : BOOL; (* Input for stopping the process *)
        FruitSelected : BOOL; (* Input indicating fruit selection *)
    END_VAR

    VAR_OUTPUT
        JuiceProcessing : BOOL; (* Output for controlling juice extraction *)
        BottleFilling : BOOL; (* Output for controlling bottle filling *)
        CapPlacement : BOOL; (* Output for placing caps on bottles *)
        Packaging : BOOL; (* Output for packaging filled bottles *)
        ProcessInProgress : BOOL; (* Indicator for an ongoing process *)
    END_VAR

    VAR
        StartRisingEdge : BOOL;
        PrevStartButton : BOOL;
    END_VAR

    (* Rising edge detection for StartButton *)
    StartRisingEdge := StartButton AND NOT PrevStartButton;
    PrevStartButton := StartButton;

    (* Process state control *)
    IF StartRisingEdge AND FruitSelected AND NOT ProcessInProgress THEN
        ProcessInProgress := TRUE;
    END_IF;

    IF StopButton OR NOT FruitSelected THEN
        ProcessInProgress := FALSE;
    END_IF;

    (* Concurrent stage outputs *)
    JuiceProcessing := ProcessInProgress;
    BottleFilling := ProcessInProgress;
    CapPlacement := ProcessInProgress;
    Packaging := ProcessInProgress;
END_FUNCTION_BLOCK;

(* ---- med_87.st ---- *)
FUNCTION_BLOCK WaterDesalination
VAR_INPUT
    StartButton : BOOL; (* Input for starting the desalination process *)
    StopButton : BOOL; (* Input for stopping the desalination process *)
    SalinitySensor : REAL; (* Input for salinity level measurement *)
END_VAR

VAR_OUTPUT
    SeawaterInletValve : BOOL; (* Output for seawater inlet valve control *)
    FreshwaterOutletValve : BOOL; (* Output for freshwater outlet valve control *)
    DesalinationInProgress : BOOL; (* Indicator for an ongoing desalination process *)
END_VAR

VAR
    MaxSalinity : REAL := 35.0; (* Maximum allowable salinity in ppm for freshwater *)
    SalinityControlSeconds : INT := 0; (* Timer for salinity control in seconds *)
END_VAR

(* Main logic body begins here *)
IF StartButton AND NOT DesalinationInProgress THEN
    SeawaterInletValve := TRUE;
    FreshwaterOutletValve := TRUE;
    DesalinationInProgress := TRUE;
    SalinityControlSeconds := 0;
ELSIF StopButton THEN
    SeawaterInletValve := FALSE;
    FreshwaterOutletValve := FALSE;
    DesalinationInProgress := FALSE;
    SalinityControlSeconds := 0;
END_IF;

IF DesalinationInProgress THEN
    SalinityControlSeconds := SalinityControlSeconds + 1;
    IF SalinityControlSeconds >= 10 THEN
        IF SalinitySensor > MaxSalinity THEN
            FreshwaterOutletValve := FALSE;
        ELSE
            FreshwaterOutletValve := TRUE;
        END_IF;
        SalinityControlSeconds := 0;
    END_IF;
END_IF;
END_FUNCTION_BLOCK;

(* ---- med_88.st ---- *)
FUNCTION_BLOCK SmartLockerControl
VAR_INPUT
    AccessCode : INT; (* Input for user access code *)
    LockerNumber : INT; (* Input for selected locker number *)
END_VAR

VAR_OUTPUT
    LockerOpen : BOOL; (* Output to control locker door *)
END_VAR

VAR
    LockerStatus : ARRAY[1..10] OF BOOL; (* Status of individual lockers: TRUE=locked, FALSE=empty *)
    LockerAccessCode : ARRAY[1..10] OF INT; (* Locker access codes *)
    bInitDone : BOOL := FALSE; (* Initialization flag *)
    i : INT; (* Loop counter - declared but not used in final implementation *)
END_VAR

(* Initialization - runs only once *)
IF NOT bInitDone THEN
    (* Initialize access codes *)
    LockerAccessCode[1] := 1234;
    LockerAccessCode[2] := 5678;
    LockerAccessCode[3] := 9876;
    LockerAccessCode[4] := 4321;
    LockerAccessCode[5] := 6543;
    LockerAccessCode[6] := 7890;
    LockerAccessCode[7] := 3456;
    LockerAccessCode[8] := 8765;
    LockerAccessCode[9] := 2345;
    LockerAccessCode[10] := 6789;

    (* Initialize all lockers to locked state (TRUE = occupied/locked) *)
    FOR i := 1 TO 10 DO
        LockerStatus[i] := TRUE;
    END_FOR;

    bInitDone := TRUE;
END_IF;

(* Main access control logic *)
LockerOpen := FALSE; (* Reset output each scan cycle *)

IF (LockerNumber >= 1) AND (LockerNumber <= 10) THEN
    IF AccessCode = LockerAccessCode[LockerNumber] THEN
        LockerOpen := TRUE;
        LockerStatus[LockerNumber] := FALSE; (* Set locker to empty/unlocked *)
    END_IF;
END_IF;

END_FUNCTION_BLOCK;

(* ---- med_89.st ---- *)
FUNCTION_BLOCK SoilTestingDeviceControl
VAR_INPUT
    StartButton : BOOL; (* Input for starting the testing process *)
    SoilSampleDetected : BOOL; (* Input for detecting soil sample *)
END_VAR

VAR_OUTPUT
    NutrientPump : BOOL; (* Output to control nutrient pump *)
    pHAdjustmentPump : BOOL; (* Output to control pH adjustment pump *)
END_VAR

VAR
    pHSensorValue : REAL; (* Simulated pH sensor value *)
    NutrientSensorValue : REAL; (* Simulated nutrient sensor value *)
    TestingStatus : INT; (* Status: 0=Idle, 1=Testing, 2=Completed *)
    NutrientThreshold : REAL := 0.7; (* Nutrient level threshold for analysis *)
    pHThreshold : REAL := 6.5; (* pH level threshold for analysis *)
END_VAR

CASE TestingStatus OF
    0: (* Idle State *)
        pHSensorValue := 7.0;
        NutrientSensorValue := 0.5;
        NutrientPump := FALSE;
        pHAdjustmentPump := FALSE;

        IF StartButton THEN
            TestingStatus := 1;
            NutrientPump := TRUE;
            pHAdjustmentPump := TRUE;
        END_IF;

    1: (* Testing State *)
        (* First check for completion conditions *)
        IF SoilSampleDetected THEN
            IF (NutrientSensorValue >= NutrientThreshold) AND (pHSensorValue <= pHThreshold) THEN
                TestingStatus := 2;
                NutrientPump := FALSE;
                pHAdjustmentPump := FALSE;
            END_IF;
        END_IF;

        (* Only update sensor values if still in Testing state *)
        IF TestingStatus = 1 THEN
            (* Update NutrientSensorValue with upper limit *)
            NutrientSensorValue := NutrientSensorValue + 0.1;
            IF NutrientSensorValue > 0.9 THEN
                NutrientSensorValue := 0.9;
            END_IF;

            (* Update pHSensorValue with lower limit *)
            pHSensorValue := pHSensorValue - 0.5;
            IF pHSensorValue < 4.0 THEN
                pHSensorValue := 4.0;
            END_IF;
        END_IF;

    2: (* Completed State *)
        NutrientPump := FALSE;
        pHAdjustmentPump := FALSE;

        (* Stay in Completed state - requires external reset *)
        (* To reset, set TestingStatus := 0 from outside *)

    ELSE
        (* Default case - reset to Idle state *)
        TestingStatus := 0;
END_CASE;

END_FUNCTION_BLOCK;

(* ---- med_90.st ---- *)
FUNCTION_BLOCK SushiConveyorControl
VAR_INPUT
    StartButton : BOOL;
    StopButton : BOOL;
    EmergencyStop : BOOL;
END_VAR

VAR_OUTPUT
    ConveyorMotor : BOOL;
END_VAR

VAR
    BeltRunning : BOOL;
    ConveyorTimer : INT;
    RotationTime : INT := 5;
END_VAR

IF EmergencyStop THEN
    ConveyorMotor := FALSE;
    BeltRunning := FALSE;
    ConveyorTimer := 0;
    RETURN;
END_IF;

IF NOT BeltRunning AND StartButton THEN
    ConveyorMotor := TRUE;
    BeltRunning := TRUE;
    ConveyorTimer := 0;
ELSIF BeltRunning AND StopButton THEN
    ConveyorMotor := FALSE;
    BeltRunning := FALSE;
    ConveyorTimer := 0;
END_IF;

IF BeltRunning THEN
    ConveyorTimer := ConveyorTimer + 1;
    IF ConveyorTimer >= RotationTime THEN
        ConveyorTimer := 0;
    END_IF;
END_IF;

END_FUNCTION_BLOCK;

(* ---- med_91.st ---- *)
FUNCTION_BLOCK AGVControlSystem
VAR_INPUT
    MaterialRequest : INT; (* New material handling request *)
END_VAR

VAR_OUTPUT
    AGV1_Ready : BOOL := TRUE; (* AGV 1 ready status *)
    AGV2_Ready : BOOL := TRUE; (* AGV 2 ready status *)
    AGV3_Ready : BOOL := TRUE; (* AGV 3 ready status *)
END_VAR

VAR
    MaterialQueue : ARRAY[1..10] OF INT; (* Material handling request queue *)
    AGVPosition : ARRAY[1..3] OF INT; (* AGV position array *)
    QueueHead : INT := 1; (* Head pointer for FIFO queue *)
    QueueTail : INT := 1; (* Tail pointer for FIFO queue *)
    QueueCount : INT := 0; (* Current number of tasks in queue *)
    AGVTask : ARRAY[1..3] OF INT := [0,0,0]; (* Current task assigned to each AGV *)
    AGVWorking : ARRAY[1..3] OF BOOL := [FALSE,FALSE,FALSE]; (* Working status of each AGV *)
    TaskToAssign : INT; (* Task to be assigned from queue *)
    Assigned : BOOL; (* Flag indicating task assignment occurred *)
    i : INT; (* Loop counter *)
    j : INT; (* Loop counter *)
    k : INT; (* Loop counter *)
END_VAR

(* 1. Queue Management: Enqueue new material requests *)
IF MaterialRequest > 0 THEN
    IF QueueCount < 10 THEN
        MaterialQueue[QueueTail] := MaterialRequest;
        QueueTail := QueueTail + 1;
        IF QueueTail > 10 THEN
            QueueTail := 1;
        END_IF;
        QueueCount := QueueCount + 1;
    END_IF;
END_IF;

(* 2. AGV Status Control: Update positions and reset upon completion *)
FOR i := 1 TO 3 DO
    IF AGVWorking[i] THEN
        AGVPosition[i] := AGVPosition[i] - 1;
        IF AGVPosition[i] <= 0 THEN
            AGVPosition[i] := 0;
            AGVWorking[i] := FALSE;
            AGVTask[i] := 0;
        END_IF;
    END_IF;
END_FOR;

(* 3. Priority-based Task Assignment: AGV1 > AGV2 > AGV3 *)
Assigned := FALSE;
IF QueueCount > 0 THEN
    TaskToAssign := MaterialQueue[QueueHead];
    FOR j := 1 TO 3 DO
        IF NOT AGVWorking[j] AND NOT Assigned THEN
            AGVWorking[j] := TRUE;
            AGVTask[j] := TaskToAssign;
            AGVPosition[j] := 10;
            QueueHead := QueueHead + 1;
            IF QueueHead > 10 THEN
                QueueHead := 1;
            END_IF;
            QueueCount := QueueCount - 1;
            Assigned := TRUE;
        END_IF;
    END_FOR;
END_IF;

(* 4. Safety Constraints: Ensure non-negative positions *)
FOR k := 1 TO 3 DO
    IF AGVPosition[k] < 0 THEN
        AGVPosition[k] := 0;
    END_IF;
END_FOR;

(* 5. State Monitoring: Update AGV ready status outputs *)
AGV1_Ready := NOT AGVWorking[1];
AGV2_Ready := NOT AGVWorking[2];
AGV3_Ready := NOT AGVWorking[3];

END_FUNCTION_BLOCK;
